Fanuc KAREL source: test_math.kl

PROGRAM test_math
%NOLOCKGROUP

VAR
  entry : INTEGER
  status : INTEGER
  -- randarr : ARRAY[200] OF REAL

%include math.klt
%include display.c.klt

%from strings.klh %import s_to_rarr, s_to_iarr, s_to_vec
%from display.klh %import clear, show
%include kunit.klh
%include math.klh

ROUTINE t_pow : BOOLEAN
  BEGIN
    RETURN(kunit_eq_r(256, math__pow(2, 8)) AND kunit_eq_r(3, math_decimal(math__pow(M_E, ln(3)), 1) ) AND
          kunit_eq_r(1, math__pow(1, M_E)) AND kunit_eq_r(70.0, math_decimal(math__pow(8.3666, 2), 1)))
  END t_pow

ROUTINE t_floor : BOOLEAN
  BEGIN
    RETURN(kunit_eq_int(3, math__floor(M_PI)) AND kunit_eq_int(-3, math__floor(-2.5)))
  END t_floor

ROUTINE t_ceil : BOOLEAN
  BEGIN
    RETURN(kunit_eq_int(4, math__ceil(M_PI)) AND kunit_eq_int(-2, math__ceil(-2.5)))
  END t_ceil

ROUTINE t_round : BOOLEAN
  BEGIN
    RETURN(kunit_eq_r(3.142, math_decimal(M_PI, 3)) AND kunit_eq_r(-6.70, math_decimal(-6.6982, 2)))
  END t_round

ROUTINE t_log10 : BOOLEAN
  BEGIN
    RETURN(kunit_eq_r(0, math__log10(1)) AND kunit_eq_r(3, math__log10(1000)) AND
           kunit_eq_r(1.69897, math__log10(50)))
  END t_log10

ROUTINE t_log2 : BOOLEAN
  BEGIN
    RETURN(kunit_eq_r(2, math__log2(4)) AND kunit_eq_r(6, math__log2(64)) AND
           kunit_eq_r(2.321928, math__log2(5)))
  END t_log2

ROUTINE t_rand : BOOLEAN
  VAR
    s_tme  : STRING[16]
    tme1, tme2, tme3, tme4 : INTEGER
    b1, b2, b3, b4 : BOOLEAN
  BEGIN
    s_tme = '02-FEB-20 01:00'
    CNV_STR_TIME(s_tme, tme1)
    math__srand(tme1)
    b1 = kunit_eq_r(0.781, math__rand)

    s_tme = '02-FEB-20 02:00'
    CNV_STR_TIME(s_tme, tme2)
    math__srand(tme2)
    b2 = kunit_eq_r(0.437, math__rand)

    s_tme = '02-FEB-20 03:00'
    CNV_STR_TIME(s_tme, tme3)
    math__srand(tme3)
    b3 = kunit_eq_r(0.093, math__rand)

    s_tme = '02-FEB-20 04:00'
    CNV_STR_TIME(s_tme, tme4)
    math__srand(tme4)
    b4 = kunit_eq_r(0.750, math__rand)

    RETURN(b1 AND b2 AND b3 AND b4)
  END t_rand

ROUTINE t_map : BOOLEAN
  BEGIN
    RETURN(kunit_eq_r(500, math__map_real(0.5, 0, 1, 0, 1000)) AND &
           kunit_eq_r(M_PI_2, math__map_real(M_PI, 0, M_PI, 0, M_PI_2)) AND &
           kunit_eq_r(2.441, math__map_real(1000, 0, math__pow(2, 11), 0, 5)) AND &
           kunit_eq_int(50, math__map_int(0.5, 0, 1, 0, 100)) AND &
           kunit_eq_int(127, math__map_int(512, 0, 1023, 0, 255)) )
  END t_map

ROUTINE t_rand_int : BOOLEAN
  VAR
    s_tme  : STRING[16]
    tme1, tme2, tme3, tme4 : INTEGER
    b1, b2, b3, b4 : BOOLEAN
  BEGIN
    s_tme = '02-FEB-20 01:00'
    CNV_STR_TIME(s_tme, tme1)
    math__srand(tme1)
    b1 = kunit_eq_int(25601, math__rand_int)

    s_tme = '02-FEB-20 02:00'
    CNV_STR_TIME(s_tme, tme2)
    math__srand(tme2)
    b2 = kunit_eq_int(14337, math__rand_int)

    s_tme = '02-FEB-20 03:00'
    CNV_STR_TIME(s_tme, tme3)
    math__srand(tme3)
    b3 = kunit_eq_int(23, math__rand_color)

    s_tme = '02-FEB-20 04:00'
    CNV_STR_TIME(s_tme, tme4)
    math__srand(tme4)
    b4 = kunit_eq_int(191, math__rand_color)

    RETURN(b1 AND b2 AND b3 AND b4)

  END t_rand_int

ROUTINE t_rand_arr : BOOLEAN
  VAR
    i    : INTEGER
    s_tme  : STRING[16]
    tme : INTEGER
    arr, sol_arr : ARRAY[10] OF REAL
  BEGIN
    s_tme = '02-FEB-20 20:20'
    CNV_STR_TIME(s_tme, tme)

    math__rand_rarr(tme, arr)

    s_to_rarr('0.08,0.667,0.414,0.454,0.292,0.039,0.829,0.917,0.664,0.204',',', sol_arr)

    RETURN(kunit_eq_arr(sol_arr, arr))
  END t_rand_arr

ROUTINE t_rand_pos : BOOLEAN
  VAR
    i    : INTEGER
    s_tme  : STRING[16]
    tme : INTEGER
    pos, sol_pos : XYZWPR
  BEGIN
    s_tme = '02-FEB-20 20:20'
    CNV_STR_TIME(s_tme, tme)

    pos = math__rand_position(tme)

    sol_pos.x = 24.038 ; sol_pos.y = 200.092 ; sol_pos.z = 124.216 ;
    sol_pos.w = 40.929 ; sol_pos.p = 26.31 ; sol_pos.r = 3.547 ;

    RETURN(kunit_eq_pos(sol_pos, pos))
  END t_rand_pos


ROUTINE t_sum : BOOLEAN
  VAR
    i    : INTEGER
    s_tme  : STRING[16]
    tme : INTEGER
    arr1 : ARRAY[10] OF REAL
    sum   : REAL
  BEGIN
    s_tme = '02-FEB-20 20:20'
    CNV_STR_TIME(s_tme, tme)
    FOR i=1 TO ARRAY_LEN(arr1) DO
      math__srand(tme*i)
      arr1[i] = ABS(math__rand)
    ENDFOR
    sum = math__sum_real(arr1)
    RETURN(kunit_eq_r(4.564, sum))
  END t_sum


ROUTINE t_count_even : BOOLEAN
  VAR
    i    : INTEGER
    arr1 : ARRAY[10] OF REAL
    sum   : REAL
  BEGIN
    FOR i=1 TO ARRAY_LEN(arr1) DO
      arr1[i] = i MOD 2
    ENDFOR
    sum = math__sum_real(arr1)
    RETURN(kunit_eq_r(5, sum))
  END t_count_even


ROUTINE t_average : BOOLEAN
  VAR
    i    : INTEGER
    arr1 : ARRAY[10] OF REAL
    ave   : REAL
  BEGIN
    FOR i=1 TO ARRAY_LEN(arr1) DO
      arr1[i] = i
    ENDFOR

    ave = math__average_real(arr1)
    RETURN(kunit_eq_r(5.5, ave))
  END t_average

ROUTINE t_ave_uninit : BOOLEAN
  VAR
    i    : INTEGER
    arr1 : ARRAY[10] OF REAL
    ave   : REAL
  BEGIN
    FOR i=1 TO ARRAY_LEN(arr1) DO
      --only insert values every other value
      IF (i MOD 2 = 0) THEN
        arr1[i] = i
      ENDIF
    ENDFOR

    ave = math__average_real(arr1)
    RETURN(kunit_eq_r(6.0, ave))
  END t_ave_uninit

ROUTINE t_matmul : BOOLEAN
  VAR
    origin : XYZWPR
    expected1, expected2, expected3  : XYZWPR
    pos1 : XYZWPR
    v1, v2 : VECTOR
  BEGIN
    origin.x = 0 ; origin.y = 0 ; origin.z = 0 ;
    origin.w = 90 ; origin.p = 0 ; origin.r = 90 ;

    --expected1
    --rotate -30 deg in w and then translate 300 in y
    expected1.x =  -150.0 ; expected1.y = 0 ; expected1.z = 259.808 ;
    expected1.w = 60 ; expected1.p = 0 ; expected1.r = 90 ;
    --translate1
    v1.x = 0 ; v1.y = 300 ; v1.z = 0 ;

    --expected2
    --rotate 90 in r, -45 in p, translate 200mm in z and -150mm in x,
    --then reverse z rotation
    expected2.x =  35.355 ; expected2.y = 0 ; expected2.z = -247.487 ;
    expected2.w = 135 ; expected2.p = 0 ; expected2.r = 90 ;
    --translate2
    v2.x = -150 ; v2.y = 0 ; v2.z = 200 ;

    --rotate 45, 90, then 180 in x,y,z respectively
    expected3.x =  0 ; expected3.y = 0 ; expected3.z = 0 ;
    expected3.w = -90 ; expected3.p = 45 ; expected3.r = 0 ;

    pos1 = math__rotz(math__roty(math__rotx((origin), 45), 90), 180)

    --display__clear
    --WRITE TPDISPLAY(CR,p_to_s(pos1))
    --display__show

  RETURN(kunit_eq_pos(origin, math__rotz(math__roty(math__roty(math__rotz((origin), 20), 45), -45), -20)) AND &
         kunit_eq_pos(expected1, math__translate(math__rotx((origin), -30), v1)) AND &
         kunit_eq_pos(expected2, math__rotz(math__translate(math__roty(math__rotz((origin), 90), -45), v2), -90)) AND &
         kunit_eq_pos(expected3, math__rotz(math__roty(math__rotx((origin), 45), 90), 180)) )
  END t_matmul


ROUTINE t_norm : BOOLEAN
  VAR
    v1, v2 : VECTOR
  BEGIN
    v1.x = 2; v1.y = -1; v1.z = -5;
    v2.x = 4; v2.y = -3; v2.z = 1;

    RETURN( kunit_eq_r(3.7417, math__norm(s_to_vec('-3,2,1',',')) ) AND &
            kunit_eq_r(6.6332, math__norm(v2-v1)) )
  END t_norm

ROUTINE t_sort : BOOLEAN
  VAR
    arr1, exp1 : ARRAY[10] OF INTEGER
    arr2, exp2 : ARRAY[10] OF REAL

    s_tme : STRING[14]
    tme : INTEGER
  BEGIN
    --populate and sort
    s_to_iarr('99,73,81,17,89,85,44,36,51,6',',',arr1)
    math__quicksort_int(arr1)

    s_to_rarr('17.75,65.77,96.02,27.65,25.22,3.04,13.53,28.45,49.12,69.72',',',arr2)
    math__quicksort_real(arr2)

    --expected
    s_to_iarr('6,17,36,44,51,73,81,85,89,99',',',exp1)
    s_to_rarr('3.04,13.53,17.75,25.22,27.65,28.45,49.12,65.77,69.72,96.02',',',exp2)

    --test overflow
    --get random real array
    -- s_tme = '10-DEC-20 8:00'
    -- CNV_STR_TIME(s_tme, tme)
    -- math__rand_rarr(tme, randarr)
    -- math__quicksort_real(randarr)

    RETURN( kunit_eq_ari(exp1, arr1) AND kunit_eq_arr(exp2, arr2) )
  END t_sort

BEGIN
  --asserts 43
  -- 18 tests
  kunit_test('test_power()', t_pow) --assert 4
  kunit_test('test_floor()', t_floor) --assert 2
  kunit_test('test_ceiling()', t_ceil) --assert 2
  kunit_test('test_rounding()', t_round) --assert 2
  kunit_test('test_log10()', t_log10) -- assert 3
  kunit_test('test_log2()', t_log2) -- assert 3
  kunit_test('test random number', t_rand) --assert 4
  kunit_test('test map function', t_map) -- assert 5
  kunit_test('test random integers', t_rand_int) --assert 4
  kunit_test('test random array', t_rand_arr) -- assert 1
  kunit_test('test random position', t_rand_pos) -- assert 1
  kunit_test('test sum of rand', t_sum) -- assert 1
  kunit_test('test count even numbers', t_count_even) -- assert 1
  kunit_test('test average numbers', t_average) -- assert 1
  kunit_test('test average uninitialized array',t_ave_uninit) -- assert 1
  kunit_test('test maxtrix multiplication', t_matmul) -- assert 4
  kunit_test('test vector norm', t_norm) --assert 2
  kunit_test('test sorting', t_sort) --assert 2

  kunit_done
END test_math
